FUNCTION_BLOCK FB_TestableGCModule EXTENDS FB_GC_Module

SUPER^();

METHOD M_SetTestServiceStatus
VAR_INPUT
	TestStatus : ST_GC_ServiceStatus;
END_VAR
_ServiceStatusView.ByName := TestStatus;
END_METHOD

METHOD M_UpdateTestAlarmList
H_UpdateAlarmList();
END_METHOD

METHOD M_SetTestSingleProcessStatus
VAR_INPUT
	TestStatus : ST_GCSingleProcessStatus;
END_VAR
_SingleProcessStatus := TestStatus;
END_METHOD

METHOD M_UpdateTestServiceDataList
H_UpdateServiceDataList();
END_METHOD

END_FUNCTION_BLOCK

(* stored: Version 1.1.0.1, ProductVersion 3.1.4026.18
   POU FB_TestableGCModule: Id {9c2f828e-112b-4c5e-8dde-b427c89f8b11}, SpecialFunc None
   Method M_SetTestServiceStatus: Id {9c2f828e-112b-4c5e-8dde-b427c89f8b12}
   Method M_UpdateTestAlarmList: Id {9c2f828e-112b-4c5e-8dde-b427c89f8b13}
   Method M_SetTestSingleProcessStatus: Id {9c2f828e-112b-4c5e-8dde-b427c89f8b14}
   Method M_UpdateTestServiceDataList: Id {9c2f828e-112b-4c5e-8dde-b427c89f8b15} *)
